// TIA Portal V20 export
// export: Created 2025-12-01T14:56:53.5824208Z, ExportSetting None, DisplayName Totally Integrated Automation Portal, DisplayVersion V20 Update 3, DisplayName TIA Portal Openness, DisplayVersion V20 Update 3, DisplayName TIA Portal Version Control Interface, DisplayVersion V20 Update 3, DisplayName STEP 7 Professional, DisplayVersion V20 Update 3, DisplayName STEP 7 Safety, DisplayVersion V20 Update 2, DisplayName WinCC Basic/Comfort/Advanced, DisplayVersion V20 Update 3, DisplayName WinCC Professional, DisplayVersion V20 Update 3, DisplayName WinCC Unified, DisplayVersion V20 Update 3
FUNCTION_BLOCK "FB481_Interlock_RIANTICS"   // FB481, LAD
{ S7_Optimized_Access := 'FALSE' }
// stored: AutoNumber false, SetENOAutomatically false
   VAR_INPUT
      Estado_CBx { ExternalVisible := 'False'; ExternalWritable := 'False'} : "EstadoZona";   // Dirección inicio periferia
      Dir_Inicial { ExternalVisible := 'False'} : UInt;
      Zona_PEPA : Bool;
      Nodo_OK : Bool;
      Activa_L1 : Bool;
      Activa_L2 : Bool;
      AVTF_PilaPequeña_L1 { ExternalVisible := 'False'} : Bool;
      AVTF_PilaGrande_L1 { ExternalVisible := 'False'} : Bool;
      Mesa_L1 : UInt;
      AVTF_Entrada_L1 { ExternalVisible := 'False'} : Bool;
      ForzarFin_Entrada_L1 : Bool;
      PTF_Salida_L1 { ExternalVisible := 'False'} : Bool;
      Mesa_L2 : UInt;
      AVTF_Entrada_L2 { ExternalVisible := 'False'} : Bool;
      ForzarFin_Entrada_L2 : Bool;
      PTF_Salida_L2 { ExternalVisible := 'False'} : Bool;
   END_VAR
   VAR_OUTPUT
      PTF_PilaPequeñaL1 : Bool;
      PTF_PilaGrande_L1 : Bool;
      PTF_Entrada_L1 : Bool;
      FTF_Entrada_L1 : Bool;
      PTF_Entrada_L2 : Bool;
      FTF_Entrada_L2 : Bool;
      AVTF_Salida_L1 : Bool;
      AVTF_Salida_L2 : Bool;
   END_VAR
   VAR_IN_OUT
      Estado_Mesa : "EstadosMesa";
   END_VAR
   VAR
      Qubiqa_Ulma { S7_SetPoint := 'True'} : "Interlock_QubiqaUlma";
      ULMA_Qubiqa { S7_SetPoint := 'True'} : "InterlocK_UlmaQubiqa";
      MEM_Entrada_L1 : Bool;
      Orden_ForzarFin_L1 : Bool;
      MEM_ForzarFin_L1 : Bool;
      MFP_ForzarFin_L1 : Bool;
      MEM_Entrada_L2 : Bool;
      Orden_ForzarFin_L2 : Bool;
      MEM_ForzarFin_L2 : Bool;
      MFP_ForzarFin_L2 : Bool;
   END_VAR
   VAR_TEMP
      Interlock_Entradas : "Interlock_QubiqaUlma";
      Interlock_Salidas : "InterlocK_UlmaQubiqa";
      P_Entradas : Any;
      P_Salidas : Any;
      P_DI_Entradas : Any;
      P_DI_Salidas : Any;
      P_L_Entradas : Any;
      P_L_Salidas : Any;
      Guardar_AR1 : DWord;
      DBInstancia : UInt;
      Numero_UT01 : UInt;
      Numero_UT02 : UInt;
      ReturnValor : Int;
      Cero : Byte;
   END_VAR
   VAR_TEMP   // added for the SCL form of the ladder/FBD networks
      _w1 : Bool;
      _w2 : Bool;
   END_VAR
BEGIN

NETWORK
TITLE = Preparacion de Punteros ANY
//////////////////////////////////////////////////////////////////////////////
/// Inicializar las variables que necesita la FB

      TAR1  #Guardar_AR1;

      L     DINO;  // Numero del DB de Instancia
      T     #DBInstancia;


//////////////////////////////////////////////////////////////////////////////
/// Puntero Any a las Entradas y Salidas (Temporales)

      LAR1  P##P_L_Entradas;  // - Any - Entradas del interlock
      L     B#16#10;  //   10H para S7
      T     LB [AR1, P#0.0];
      L     B#16#2;  //   Tipo de Datos (BYTE)
      T     LB [AR1, P#1.0];
      L     66;  //   Cantidad de datos a leer 66 Bytes
      T     LW [AR1, P#2.0];
      L     0;  //   Numero de DB (Temporal = 0)
      T     LW [AR1, P#4.0];
      L     P##Interlock_Entradas;  //   Direccion de Inicio
      T     LD [AR1, P#6.0];
      L     B#16#87;  //   El Area de Memoria = Temporal (Nota: No 86)
      T     LB [AR1, P#6.0];


      LAR1  P##P_L_Salidas;  // - Any - Salidas del interlock
      L     B#16#10;  //   10H para S7
      T     LB [AR1, P#0.0];
      L     B#16#2;  //   Tipo de Datos (BYTE)
      T     LB [AR1, P#1.0];
      L     66;  //   Cantidad de datos a leer 66 Bytes
      T     LW [AR1, P#2.0];
      L     0;  //   Numero de DB (Temporal = 0)
      T     LW [AR1, P#4.0];
      L     P##Interlock_Salidas;  //   Direccion de Inicio
      T     LD [AR1, P#6.0];
      L     B#16#87;  //   El Area de Memoria = Temporal (Nota: No 86)
      T     LB [AR1, P#6.0];


//////////////////////////////////////////////////////////////////////////////
/// Puntero Any a las Entradas y Salidas (DB de Instancia)

      LAR1  P##P_DI_Entradas;  // - Any - Entradas del interlock
      L     B#16#10;  //   10H para S7
      T     LB [AR1, P#0.0];
      L     B#16#2;  //   Tipo de Datos (BYTE)
      T     LB [AR1, P#1.0];
      L     66;  //   Cantidad de datos a leer 66 Bytes
      T     LW [AR1, P#2.0];
      L     #DBInstancia;  //   Numero de DB
      T     LW [AR1, P#4.0];
      L     P##Qubiqa_Ulma;  //   Direccion de Inicio
      T     LD [AR1, P#6.0];
      L     B#16#84;  //   El Area de Memoria = DB Instancia
      T     LB [AR1, P#6.0];

      LAR1  P##P_DI_Salidas;  // - Any - Salidas del interlock
      L     B#16#10;  //   10H para S7
      T     LB [AR1, P#0.0];
      L     B#16#2;  //   Tipo de Datos (BYTE)
      T     LB [AR1, P#1.0];
      L     66;  //   Cantidad de datos a leer 66 Bytes
      T     LW [AR1, P#2.0];
      L     #DBInstancia;  //   Numero de DB (Temporal = 0)
      T     LW [AR1, P#4.0];
      L     P##ULMA_Qubiqa;  //   Direccion de Inicio
      T     LD [AR1, P#6.0];
      L     B#16#84;  //   El Area de Memoria = DB Instancia
      T     LB [AR1, P#6.0];


//////////////////////////////////////////////////////////////////////////////
/// Puntero Any - De Lectura y Escritura de QUBIQA

      LAR1  P##P_Entradas;  // - Any - Entradas del interlock
      L     B#16#10;  //   10H para S7
      T     LB [AR1, P#0.0];
      L     B#16#2;  //   Tipo de Datos (BYTE)
      T     LB [AR1, P#1.0];
      L     66;  //   Cantidad de datos a leer 66 Bytes
      T     LW [AR1, P#2.0];
      L     0;  //   Numero de DB (Temporal = 0)
      T     LW [AR1, P#4.0];
      L     #Dir_Inicial;  //   Direccion de Inicio
      SLD   3;
      T     LD [AR1, P#6.0];
      L     B#16#81;  //   El Area de Memoria = Entradas
      T     LB [AR1, P#6.0];

      LAR1  P##P_Salidas;  // - Any - Entradas del interlock
      L     B#16#10;  //   10H para S7
      T     LB [AR1, P#0.0];
      L     B#16#2;  //   Tipo de Datos (BYTE)
      T     LB [AR1, P#1.0];
      L     66;  //   Cantidad de datos a leer 66 Bytes
      T     LW [AR1, P#2.0];
      L     0;  //   Numero de DB (Temporal = 0)
      T     LW [AR1, P#4.0];
      L     #Dir_Inicial;  //   Direccion de Inicio
      SLD   3;
      T     LD [AR1, P#6.0];
      L     B#16#82;  //   El Area de Memoria = Salidas
      T     LB [AR1, P#6.0];


/////////////////////////////////////////////////////////////////////////////////

      LAR1  #Guardar_AR1;  // Recupero para Continuar



NETWORK
TITLE = Inicializacion de las Entradas y Salidas
//////////////////////////////////////////////////////////////////////////////
/// Inicializar el interlock (Variables Temporales)

      L     0;
      T     #Cero;

      CALL  FILL
      ( BVAL    := #Cero,
        RET_VAL := #ReturnValor,
        BLK     := #P_L_Entradas
      );  // Inicializo las Entradas

      CALL  FILL
      ( BVAL    := #Cero,
        RET_VAL := #ReturnValor,
        BLK     := #P_L_Salidas
      );  // Inicializo las Salidas



NETWORK
TITLE = Lectura de las Entradas
//////////////////////////////////////////////////////////////////////////////
/// Lectura de las Entradas

      SET;  // Comprobacion del Nodo
      AN    #Nodo_OK;
      JC    NoLeerInterlock;

      CALL  BLKMOV
      ( SRCBLK  := #P_Entradas,
        RET_VAL := #ReturnValor,
        DSTBLK  := #P_L_Entradas
      );


//////////////////////////////////////////////////////////////////////////////
/// Final Lectura de las Entradas

NoLeerInterlock:NOP   0;

      CALL  BLKMOV
      ( SRCBLK  := #P_L_Entradas,
        RET_VAL := #ReturnValor,
        DSTBLK  := #P_DI_Entradas
      );  // Guardar el DB de Instancia



NETWORK
TITLE = Leer datos de la UT de la Linea 01
//////////////////////////////////////////////////////////////////////////////
/// Miro si tratar la L2

      AN    #Activa_L1;
      JC    NoExiteUT_L1;

//////////////////////////////////////////////////////////////////////////////
/// Leer Datos Exitentes para la UT

      L     "DB810_ColasMesas".Colas[#Mesa_L1].UT_PrimeraMesa;

      T     #Numero_UT01;  // Primera UT de la Mesa
      L     0;
      ==I;
      JC    NoExiteUT_L1;

// Numero de Bulto
      L     "DB815_UTs_Datos".UT[#Numero_UT01].CotaAnchura;
      T     #Interlock_Salidas.ItemsNo_L1;

// Numero de Bultos (Total)
      L     "DB815_UTs_Datos".UT[#Numero_UT01].CotaProfundidad;
      T     #Interlock_Salidas.ItemsNoTotal_L1;

// Longitud del PID
      L     20;
      T     #Interlock_Salidas.Length_PID_L1;

// Copia del PID
      CALL  BLKMOV
      ( SRCBLK  := "DB814_UTs_Etiqueta".UT[#Numero_UT01].EtiquetaRouter,
        RET_VAL := #ReturnValor,
        DSTBLK  := #Interlock_Salidas.PID_L1
      );

NoExiteUT_L1:NOP   0;  // Final de la Lectura de Datos



NETWORK
TITLE = Leer datos de la UT de la Linea 02
//////////////////////////////////////////////////////////////////////////////
/// Miro si tratar la L2

      AN    #Activa_L2;
      JC    NoExiteUT_L2;

//////////////////////////////////////////////////////////////////////////////
/// Leer Datos Exitentes para la UT

      L     "DB810_ColasMesas".Colas[#Mesa_L2].UT_PrimeraMesa;
      T     #Numero_UT02;  // Primera UT de la Mesa

      L     0;
      ==I;
      JC    NoExiteUT_L2;

// Numero de Bulto
      L     "DB815_UTs_Datos".UT[#Numero_UT02].CotaAnchura;
      T     #Interlock_Salidas.ItemsNo_L2;

// Numero de Bultos (Total)
      L     "DB815_UTs_Datos".UT[#Numero_UT02].CotaProfundidad;
      T     #Interlock_Salidas.ItemsNoTotal_L2;

// Longitud del PID
      L     20;
      T     #Interlock_Salidas.Length_PID_L2;

// Copia del PID
      CALL  BLKMOV
      ( SRCBLK  := "DB814_UTs_Etiqueta".UT[#Numero_UT02].EtiquetaRouter,
        RET_VAL := #ReturnValor,
        DSTBLK  := #Interlock_Salidas.PID_L2
      );

NoExiteUT_L2:NOP   0;  // Final de la Lectura de Datos



NETWORK
TITLE = Leer Forzado de la Linea 01
//////////////////////////////////////////////////////////////////////////////
/// Leer si hay Orden de Forzado

      SET;
      R     #Orden_ForzarFin_L1;  // Inicializado el forzado

      L     "DB841_Recepcion".Mesa[#Mesa_L1].Auxiliar_04;
      L     0;
      ==I;  // Mirar si hay Forzado
      JC    NoForzado_L1;

      SET;  // Activo para realizar Forzado
      S     #Orden_ForzarFin_L1;

      L     0;  // Dar por Tratado el Forzado
      T     "DB841_Recepcion".Mesa[#Mesa_L1].Auxiliar_04;

NoForzado_L1:NOP   0;



NETWORK
TITLE = Leer Forzado de la Linea 02
//////////////////////////////////////////////////////////////////////////////
/// Leer si hay Orden de Forzado

      SET;
      R     #Orden_ForzarFin_L2;  // Inicializado el forzado

      SET;  // Esta Operativa la L2
      AN    #Activa_L2;
      JC    NoForzado_L2;

      L     "DB841_Recepcion".Mesa[#Mesa_L2].Auxiliar_04;
      L     0;
      ==I;  // Mirar si hay Forzado
      JC    NoForzado_L2;

      SET;
      S     #Orden_ForzarFin_L2;  // Activo para realizar Forzado

      L     0;  // Dar por Tratado el Forzado
      T     "DB841_Recepcion".Mesa[#Mesa_L2].Auxiliar_04;

NoForzado_L2:NOP   0;



NETWORK
TITLE = Final de la Inicializacion
//////////////////////////////////////////////////////////////////////////////
/// Final de la Inicializacion de la Funcion

      LAR1  #Guardar_AR1;


REGION Network 10: Salidas Comunes
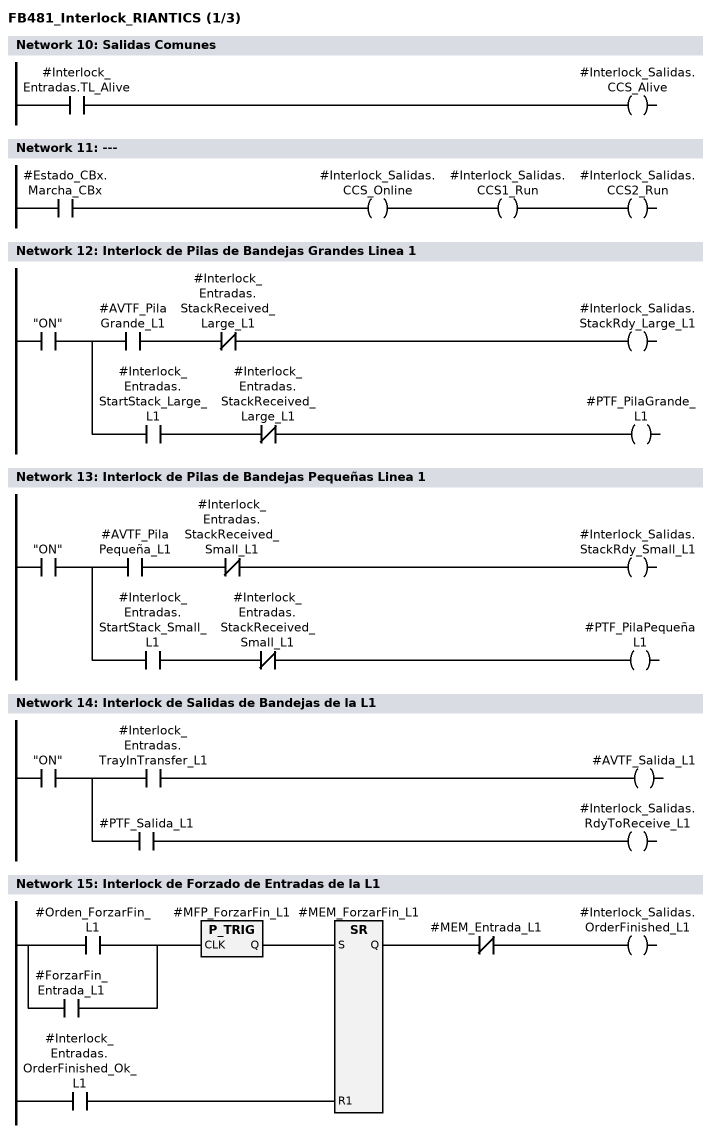
   RUNG wire#powerrail
      Contact( #Interlock_Entradas.TL_Alive )
      Coil( #Interlock_Salidas.CCS_Alive )
   END_RUNG
   // the same network as SCL:
   #Interlock_Salidas.CCS_Alive := #Interlock_Entradas.TL_Alive;
END_REGION

REGION Network 11: ---
   RUNG wire#powerrail
      Contact( #Estado_CBx.Marcha_CBx )
      Coil( #Interlock_Salidas.CCS_Online )
      Coil( #Interlock_Salidas.CCS1_Run )
      Coil( #Interlock_Salidas.CCS2_Run )
   END_RUNG
   // the same network as SCL:
   #Interlock_Salidas.CCS_Online := #Estado_CBx.Marcha_CBx;
   #Interlock_Salidas.CCS1_Run := #Estado_CBx.Marcha_CBx;
   #Interlock_Salidas.CCS2_Run := #Estado_CBx.Marcha_CBx;
END_REGION

REGION Network 12: Interlock de Pilas de Bandejas Grandes Linea 1
   RUNG wire#powerrail
      Contact( "ON" )
      wire#w1
      Contact( #AVTF_PilaGrande_L1 )
      I_Contact( #Interlock_Entradas.StackReceived_Large_L1 )
      Coil( #Interlock_Salidas.StackRdy_Large_L1 )
   END_RUNG
   RUNG wire#w1
      Contact( #Interlock_Entradas.StartStack_Large_L1 )
      I_Contact( #Interlock_Entradas.StackReceived_Large_L1 )
      Coil( #PTF_PilaGrande_L1 )
   END_RUNG
   // the same network as SCL:
   #Interlock_Salidas.StackRdy_Large_L1 := "ON" AND #AVTF_PilaGrande_L1 AND NOT #Interlock_Entradas.StackReceived_Large_L1;
   #PTF_PilaGrande_L1 := "ON" AND #Interlock_Entradas.StartStack_Large_L1 AND NOT #Interlock_Entradas.StackReceived_Large_L1;
END_REGION

REGION Network 13: Interlock de Pilas de Bandejas Pequeñas Linea 1
   RUNG wire#powerrail
      Contact( "ON" )
      wire#w1
      Contact( #AVTF_PilaPequeña_L1 )
      I_Contact( #Interlock_Entradas.StackReceived_Small_L1 )
      Coil( #Interlock_Salidas.StackRdy_Small_L1 )
   END_RUNG
   RUNG wire#w1
      Contact( #Interlock_Entradas.StartStack_Small_L1 )
      I_Contact( #Interlock_Entradas.StackReceived_Small_L1 )
      Coil( #PTF_PilaPequeñaL1 )
   END_RUNG
   // the same network as SCL:
   #Interlock_Salidas.StackRdy_Small_L1 := "ON" AND #AVTF_PilaPequeña_L1 AND NOT #Interlock_Entradas.StackReceived_Small_L1;
   #PTF_PilaPequeñaL1 := "ON" AND #Interlock_Entradas.StartStack_Small_L1 AND NOT #Interlock_Entradas.StackReceived_Small_L1;
END_REGION

REGION Network 14: Interlock de Salidas de Bandejas de la L1
   RUNG wire#powerrail
      Contact( "ON" )
      wire#w1
      Contact( #Interlock_Entradas.TrayInTransfer_L1 )
      Coil( #AVTF_Salida_L1 )
   END_RUNG
   RUNG wire#w1
      Contact( #PTF_Salida_L1 )
      Coil( #Interlock_Salidas.RdyToReceive_L1 )
   END_RUNG
   // the same network as SCL:
   #AVTF_Salida_L1 := "ON" AND #Interlock_Entradas.TrayInTransfer_L1;
   #Interlock_Salidas.RdyToReceive_L1 := "ON" AND #PTF_Salida_L1;
END_REGION

REGION Network 15: Interlock de Forzado de Entradas de la L1
   RUNG wire#powerrail
      Contact( #Orden_ForzarFin_L1 )
      wire#w1
      P_Trig( #MFP_ForzarFin_L1 )
      S_SR(operand := #MEM_ForzarFin_L1, r1 := wire#w2)
      I_Contact( #MEM_Entrada_L1 )
      Coil( #Interlock_Salidas.OrderFinished_L1 )
   END_RUNG
   RUNG wire#powerrail
      Contact( #ForzarFin_Entrada_L1 )
   END_RUNG wire#w1
   RUNG wire#powerrail
      Contact( #Interlock_Entradas.OrderFinished_Ok_L1 )
   END_RUNG wire#w2
   // the same network as SCL:
   #_w1 := #Orden_ForzarFin_L1 OR #ForzarFin_Entrada_L1;
   #_w2 := #_w1 AND NOT #MFP_ForzarFin_L1;   // rising edge
   #MFP_ForzarFin_L1 := #_w1;
   IF #_w2 THEN
       #MEM_ForzarFin_L1 := TRUE;   // SR flip-flop
   END_IF;
   IF #Interlock_Entradas.OrderFinished_Ok_L1 THEN #MEM_ForzarFin_L1 := FALSE; END_IF;
   #Interlock_Salidas.OrderFinished_L1 := #MEM_ForzarFin_L1 AND NOT #MEM_Entrada_L1;
END_REGION

REGION Network 16: Interlock de Entradas de Bultos a la L1
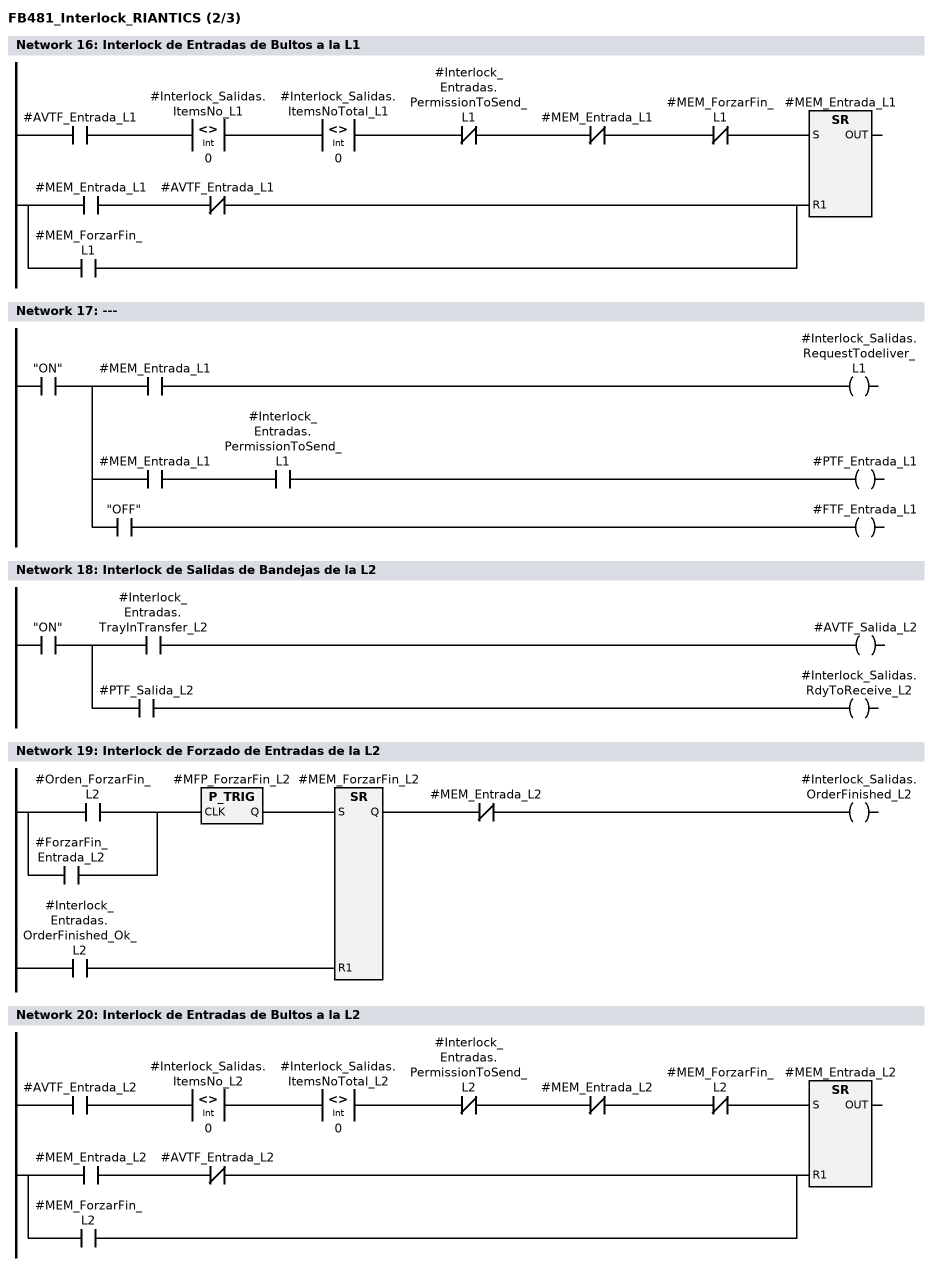
   RUNG wire#powerrail
      Contact( #AVTF_Entrada_L1 )
      { S7_Templates := "SrcType := Int" } NE_Contact(in1 := #Interlock_Salidas.ItemsNo_L1, in2 := 0)
      { S7_Templates := "SrcType := Int" } NE_Contact(in1 := #Interlock_Salidas.ItemsNoTotal_L1, in2 := 0)
      I_Contact( #Interlock_Entradas.PermissionToSend_L1 )
      I_Contact( #MEM_Entrada_L1 )
      I_Contact( #MEM_ForzarFin_L1 )
      S_SR(operand := #MEM_Entrada_L1, r1 := wire#w1)
   END_RUNG
   RUNG wire#powerrail
      Contact( #MEM_Entrada_L1 )
      I_Contact( #AVTF_Entrada_L1 )
   END_RUNG wire#w1
   RUNG wire#powerrail
      Contact( #MEM_ForzarFin_L1 )
   END_RUNG wire#w1
   // the same network as SCL:
   #_w1 := (#MEM_Entrada_L1 AND NOT #AVTF_Entrada_L1) OR #MEM_ForzarFin_L1;
   IF #AVTF_Entrada_L1 AND (#Interlock_Salidas.ItemsNo_L1 <> 0) AND (#Interlock_Salidas.ItemsNoTotal_L1 <> 0) AND NOT #Interlock_Entradas.PermissionToSend_L1 AND NOT #MEM_Entrada_L1 AND NOT #MEM_ForzarFin_L1 THEN
       #MEM_Entrada_L1 := TRUE;   // SR flip-flop
   END_IF;
   IF #_w1 THEN #MEM_Entrada_L1 := FALSE; END_IF;
END_REGION

REGION Network 17: ---
   RUNG wire#powerrail
      Contact( "ON" )
      wire#w1
      Contact( #MEM_Entrada_L1 )
      Coil( #Interlock_Salidas.RequestTodeliver_L1 )
   END_RUNG
   RUNG wire#w1
      Contact( #MEM_Entrada_L1 )
      Contact( #Interlock_Entradas.PermissionToSend_L1 )
      Coil( #PTF_Entrada_L1 )
   END_RUNG
   RUNG wire#w1
      Contact( "OFF" )
      Coil( #FTF_Entrada_L1 )
   END_RUNG
   // the same network as SCL:
   #Interlock_Salidas.RequestTodeliver_L1 := "ON" AND #MEM_Entrada_L1;
   #PTF_Entrada_L1 := "ON" AND #MEM_Entrada_L1 AND #Interlock_Entradas.PermissionToSend_L1;
   #FTF_Entrada_L1 := "ON" AND "OFF";
END_REGION

REGION Network 18: Interlock de Salidas de Bandejas de la L2
   RUNG wire#powerrail
      Contact( "ON" )
      wire#w1
      Contact( #Interlock_Entradas.TrayInTransfer_L2 )
      Coil( #AVTF_Salida_L2 )
   END_RUNG
   RUNG wire#w1
      Contact( #PTF_Salida_L2 )
      Coil( #Interlock_Salidas.RdyToReceive_L2 )
   END_RUNG
   // the same network as SCL:
   #AVTF_Salida_L2 := "ON" AND #Interlock_Entradas.TrayInTransfer_L2;
   #Interlock_Salidas.RdyToReceive_L2 := "ON" AND #PTF_Salida_L2;
END_REGION

REGION Network 19: Interlock de Forzado de Entradas de la L2
   RUNG wire#powerrail
      Contact( #Orden_ForzarFin_L2 )
      wire#w1
      P_Trig( #MFP_ForzarFin_L2 )
      S_SR(operand := #MEM_ForzarFin_L2, r1 := wire#w2)
      I_Contact( #MEM_Entrada_L2 )
      Coil( #Interlock_Salidas.OrderFinished_L2 )
   END_RUNG
   RUNG wire#powerrail
      Contact( #ForzarFin_Entrada_L2 )
   END_RUNG wire#w1
   RUNG wire#powerrail
      Contact( #Interlock_Entradas.OrderFinished_Ok_L2 )
   END_RUNG wire#w2
   // the same network as SCL:
   #_w1 := #Orden_ForzarFin_L2 OR #ForzarFin_Entrada_L2;
   #_w2 := #_w1 AND NOT #MFP_ForzarFin_L2;   // rising edge
   #MFP_ForzarFin_L2 := #_w1;
   IF #_w2 THEN
       #MEM_ForzarFin_L2 := TRUE;   // SR flip-flop
   END_IF;
   IF #Interlock_Entradas.OrderFinished_Ok_L2 THEN #MEM_ForzarFin_L2 := FALSE; END_IF;
   #Interlock_Salidas.OrderFinished_L2 := #MEM_ForzarFin_L2 AND NOT #MEM_Entrada_L2;
END_REGION

REGION Network 20: Interlock de Entradas de Bultos a la L2
   RUNG wire#powerrail
      Contact( #AVTF_Entrada_L2 )
      { S7_Templates := "SrcType := Int" } NE_Contact(in1 := #Interlock_Salidas.ItemsNo_L2, in2 := 0)
      { S7_Templates := "SrcType := Int" } NE_Contact(in1 := #Interlock_Salidas.ItemsNoTotal_L2, in2 := 0)
      I_Contact( #Interlock_Entradas.PermissionToSend_L2 )
      I_Contact( #MEM_Entrada_L2 )
      I_Contact( #MEM_ForzarFin_L2 )
      S_SR(operand := #MEM_Entrada_L2, r1 := wire#w1)
   END_RUNG
   RUNG wire#powerrail
      Contact( #MEM_Entrada_L2 )
      I_Contact( #AVTF_Entrada_L2 )
   END_RUNG wire#w1
   RUNG wire#powerrail
      Contact( #MEM_ForzarFin_L2 )
   END_RUNG wire#w1
   // the same network as SCL:
   #_w1 := (#MEM_Entrada_L2 AND NOT #AVTF_Entrada_L2) OR #MEM_ForzarFin_L2;
   IF #AVTF_Entrada_L2 AND (#Interlock_Salidas.ItemsNo_L2 <> 0) AND (#Interlock_Salidas.ItemsNoTotal_L2 <> 0) AND NOT #Interlock_Entradas.PermissionToSend_L2 AND NOT #MEM_Entrada_L2 AND NOT #MEM_ForzarFin_L2 THEN
       #MEM_Entrada_L2 := TRUE;   // SR flip-flop
   END_IF;
   IF #_w1 THEN #MEM_Entrada_L2 := FALSE; END_IF;
END_REGION

REGION Network 21: ---
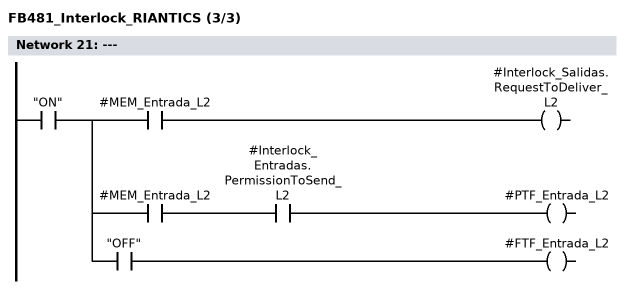
   RUNG wire#powerrail
      Contact( "ON" )
      wire#w1
      Contact( #MEM_Entrada_L2 )
      Coil( #Interlock_Salidas.RequestToDeliver_L2 )
   END_RUNG
   RUNG wire#w1
      Contact( #MEM_Entrada_L2 )
      Contact( #Interlock_Entradas.PermissionToSend_L2 )
      Coil( #PTF_Entrada_L2 )
   END_RUNG
   RUNG wire#w1
      Contact( "OFF" )
      Coil( #FTF_Entrada_L2 )
   END_RUNG
   // the same network as SCL:
   #Interlock_Salidas.RequestToDeliver_L2 := "ON" AND #MEM_Entrada_L2;
   #PTF_Entrada_L2 := "ON" AND #MEM_Entrada_L2 AND #Interlock_Entradas.PermissionToSend_L2;
   #FTF_Entrada_L2 := "ON" AND "OFF";
END_REGION

NETWORK
TITLE = Escritura de las Salidas
//////////////////////////////////////////////////////////////////////////////
/// Escritura de las Salidas

      SET;  // Comprobacion del Nodo
      AN    #Nodo_OK;
      JC    NoEscribirInterlock;

      CALL  BLKMOV
      ( SRCBLK  := #P_L_Salidas,
        RET_VAL := #ReturnValor,
        DSTBLK  := #P_Salidas
      );


//////////////////////////////////////////////////////////////////////////////
/// Final Esctitura de las Salidas

NoEscribirInterlock:NOP   0;

      CALL  BLKMOV
      ( SRCBLK  := #P_L_Salidas,
        RET_VAL := #ReturnValor,
        DSTBLK  := #P_DI_Salidas
      );  // Guardar el DB de Instancia




NETWORK
TITLE = Final de la Funcion
//////////////////////////////////////////////////////////////////////////////
/// Final de la Funcion


END_FUNCTION_BLOCK
